(* CODESYS project ExportWithApplication.export

Project tree, tasks and I/O mapping:
  application Application
    libraries: 
    task PLC_Task (cyclic, interval t#10ms, priority 14) calls PLC_PRG
    data type DUT
    program PLC_PRG [ST]: ACT, Prop
    program POU [ST]
    Symbols
*)

// Application/DUT
TYPE DUT :
STRUCT
END_STRUCT
END_TYPE

// Application/PLC_PRG
PROGRAM PLC_PRG
VAR
END_VAR

ACTION ACT:

END_ACTION

PROPERTY Prop : INT
GET
END_GET
SET
END_SET
END_PROPERTY

END_PROGRAM

// Application/POU
PROGRAM POU
VAR
END_VAR

END_PROGRAM
